# EPICS substitutions: db/ecmcEL4134.substitutions
file ecmcEcSlave.template
{
    pattern {}
            {}
}

file ecmcEL4XXX-chX.template
{
	pattern {CH_ID, LINR,    ESLO,             EOFF,   EGU,   PREC, LOW, LOLO, HIGH, HIHI, HYST, LLSV,    LSV,     HSV,     HHSV   }
		    {1,     "SLOPE", 3.0518509476E-4,  0,      "V",   3,    -10, -10,  10,   10,   0,    "MAJOR", "MINOR", "MINOR", "MAJOR"}
		    {2,     "SLOPE", 3.0518509476E-4,  0,      "V",   3,    -10, -10,  10,   10,   0,    "MAJOR", "MINOR", "MINOR", "MAJOR"}
		    {3,     "SLOPE", 3.0518509476E-4,  0,      "V",   3,    -10, -10,  10,   10,   0,    "MAJOR", "MINOR", "MINOR", "MAJOR"}
		    {4,     "SLOPE", 3.0518509476E-4,  0,      "V",   3,    -10, -10,  10,   10,   0,    "MAJOR", "MINOR", "MINOR", "MAJOR"}
}
